Fanuc KAREL source: kc00027.KL

-- PROVISIONAL review KL for V770-1; original PC SHA256 cf3eb7efdb6dc542a102203669de0f3e1fc6161dffefc2e18fc8af3572763612
-- Incomplete behavior may be omitted. Consult companion uncertainty JSON. Do not deploy.
PROGRAM KC00027
%NOLOCKGROUP
BEGIN
  -- UNRESOLVED_PC offsets 5-81; opcodes 27,22,1C,22,1C,22,1C,22,22,1C,22,22,22,31
  -- UNRESOLVED_PC offsets 86-90; opcodes 7F
END KC00027
